FUNCTION_BLOCK trip_controller_timer (* Composite Function Block Type *)
  (* Standard: 61499-2 *)
  (* Version 0.0, 11/29/2016, gulzha, nxtControl GmbH, template *)
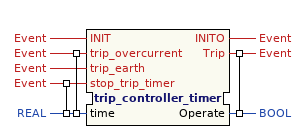
  EVENT_INPUT
    INIT; (* Initialization Request *)
    trip_overcurrent WITH time; (* Normal Execution Request *)
    trip_earth; (* Normal Execution Request *)
    stop_trip_timer WITH time;
  END_EVENT
  EVENT_OUTPUT
    INITO; (* Initialization Confirm *)
    Trip WITH Operate; (* Execution Confirmation *)
  END_EVENT
  VAR_INPUT
    time : REAL;
  END_VAR
  VAR_OUTPUT
    Operate : BOOL; (* Current Output State *)
  END_VAR
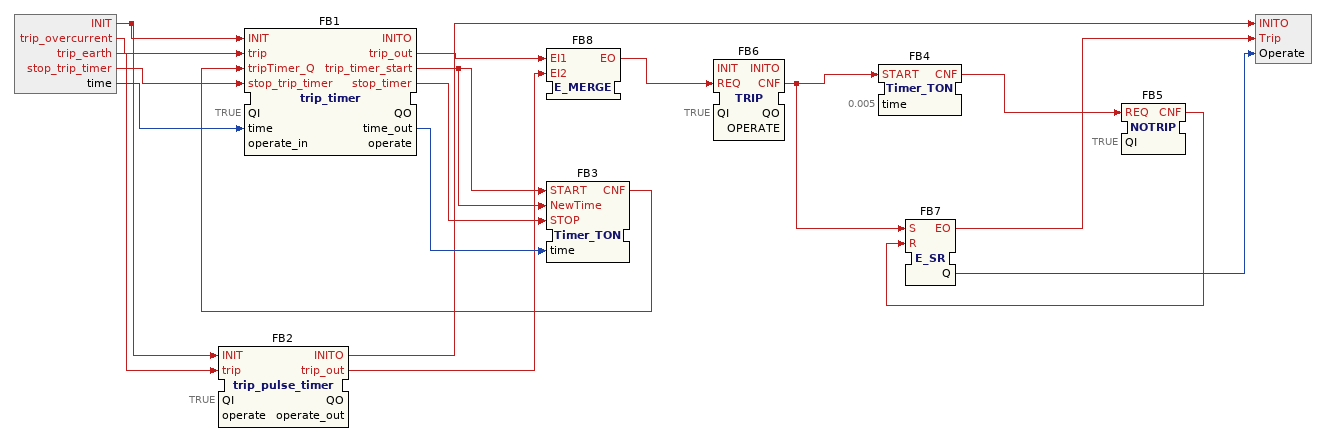
  FBS
    FB3 : Timer_TON;
    FB4 : Timer_TON(time := 0.005);
    FB5 : NOTRIP(QI := TRUE);
    FB2 : trip_pulse_timer(QI := TRUE);
    FB1 : trip_timer(QI := TRUE);
    FB6 : TRIP(QI := TRUE);
    FB8 : E_MERGE;
    FB7 : E_SR;
  END_FBS
  EVENT_CONNECTIONS
    INIT TO FB1.INIT;
    FB1.trip_timer_start TO FB3.START;
    FB1.trip_timer_start TO FB3.NewTime;
    FB1.stop_timer TO FB3.STOP;
    FB3.CNF TO FB1.tripTimer_Q;
    FB4.CNF TO FB5.REQ;
    FB1.trip_out TO FB8.EI1;
    FB2.trip_out TO FB8.EI2;
    FB8.EO TO FB6.REQ;
    FB6.CNF TO FB4.START;
    trip_overcurrent TO FB1.trip;
    trip_earth TO FB2.trip;
    INIT TO FB2.INIT;
    FB2.INITO TO INITO;
    FB6.CNF TO FB7.S;
    FB5.CNF TO FB7.R;
    FB7.EO TO Trip;
    stop_trip_timer TO FB1.stop_trip_timer;
  END_CONNECTIONS
  DATA_CONNECTIONS
    FB1.time_out TO FB3.time;
    time TO FB1.time;
    FB7.Q TO Operate;
  END_CONNECTIONS
END_FUNCTION_BLOCK
